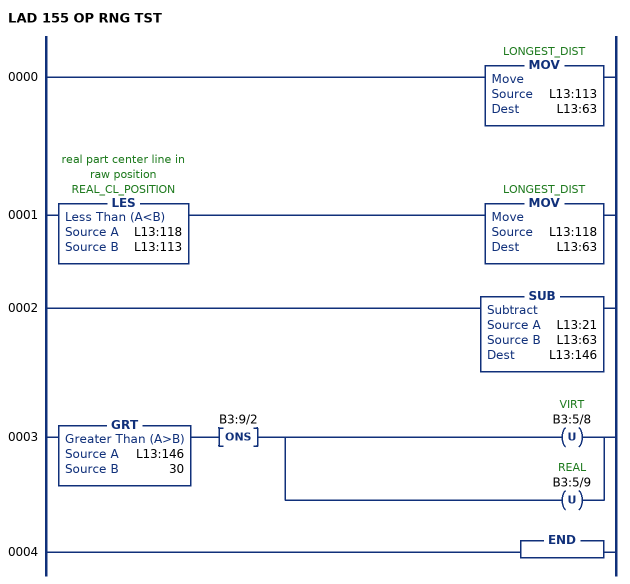
% Rung: 0 %
SOR MOV L13:113 L13:63 EOR
%   L13:113  VERTUAL_CL_POSITION  "virtual part center line transfer from the bottom in raw position" %
%   L13:63  LONGEST_DIST %
% Rung: 1 %
SOR LES L13:118 L13:113 MOV L13:118 L13:63 EOR
%   L13:118  REAL_CL_POSITION  "real part center line in raw position" %
%   L13:113  VERTUAL_CL_POSITION  "virtual part center line transfer from the bottom in raw position" %
%   L13:63  LONGEST_DIST %
% Rung: 2 %
SOR SUB L13:21 L13:63 L13:146 EOR
%   L13:21  TOP_POSITION %
%   L13:63  LONGEST_DIST %
% Rung: 3 %
SOR GRT L13:146 30 ONS B3:9/2 BST OTU B3:5/8 NXB OTU B3:5/9 BND EOR
%   B3:5/8  VIRT %
%   B3:5/9  REAL %
% Rung: 4 %
SOR END EOR

LADDER 190 "INS5"
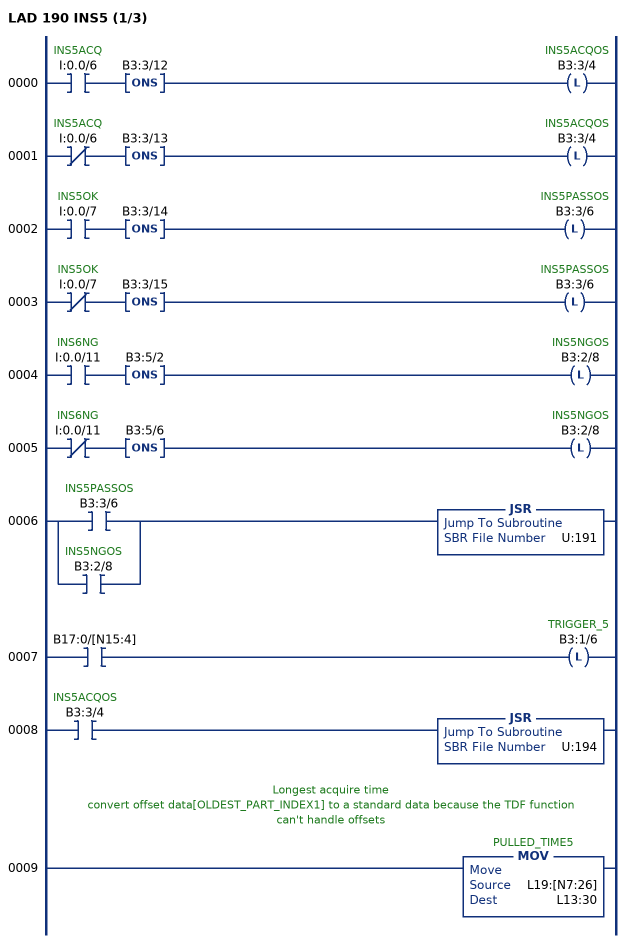
% Rung: 0 %
SOR XIC I:0.0/6 ONS B3:3/12 OTL B3:3/4 EOR
%   I:0.0/6  INS5ACQ %
%   B3:3/4  INS5ACQOS %
% Rung: 1 %
SOR XIO I:0.0/6 ONS B3:3/13 OTL B3:3/4 EOR
%   I:0.0/6  INS5ACQ %
%   B3:3/4  INS5ACQOS %
% Rung: 2 %
SOR XIC I:0.0/7 ONS B3:3/14 OTL B3:3/6 EOR
%   I:0.0/7  INS5OK %
%   B3:3/6  INS5PASSOS %
% Rung: 3 %
SOR XIO I:0.0/7 ONS B3:3/15 OTL B3:3/6 EOR
%   I:0.0/7  INS5OK %
%   B3:3/6  INS5PASSOS %
% Rung: 4 %
SOR XIC I:0.0/11 ONS B3:5/2 OTL B3:2/8 EOR
%   I:0.0/11  INS6NG %
%   B3:2/8  INS5NGOS %
% Rung: 5 %
SOR XIO I:0.0/11 ONS B3:5/6 OTL B3:2/8 EOR
%   I:0.0/11  INS6NG %
%   B3:2/8  INS5NGOS %
% Rung: 6 %
SOR BST XIC B3:3/6 NXB XIC B3:2/8 BND JSR U:191 EOR
%   B3:3/6  INS5PASSOS %
%   B3:2/8  INS5NGOS %
% Rung: 7 %
SOR XIC B17:0/[N15:4] OTL B3:1/6 EOR
%   B17:0  GOOD1 %
%   N15:4  INS_5_TRIG_LOC %
%   B3:1/6  TRIGGER_5 %
% Rung: 8 %
SOR XIC B3:3/4 JSR U:194 EOR
%   B3:3/4  INS5ACQOS %
% Rung: 9 %
% Longest acquire time
% convert offset data[OLDEST_PART_INDEX1] to a standard data because the TDF function can't handle offsets %
SOR MOV L19:[N7:26] L13:30 EOR
%   N7:26  OLDEST_PART_INDEX5 %
%   L13:30  PULLED_TIME5 %

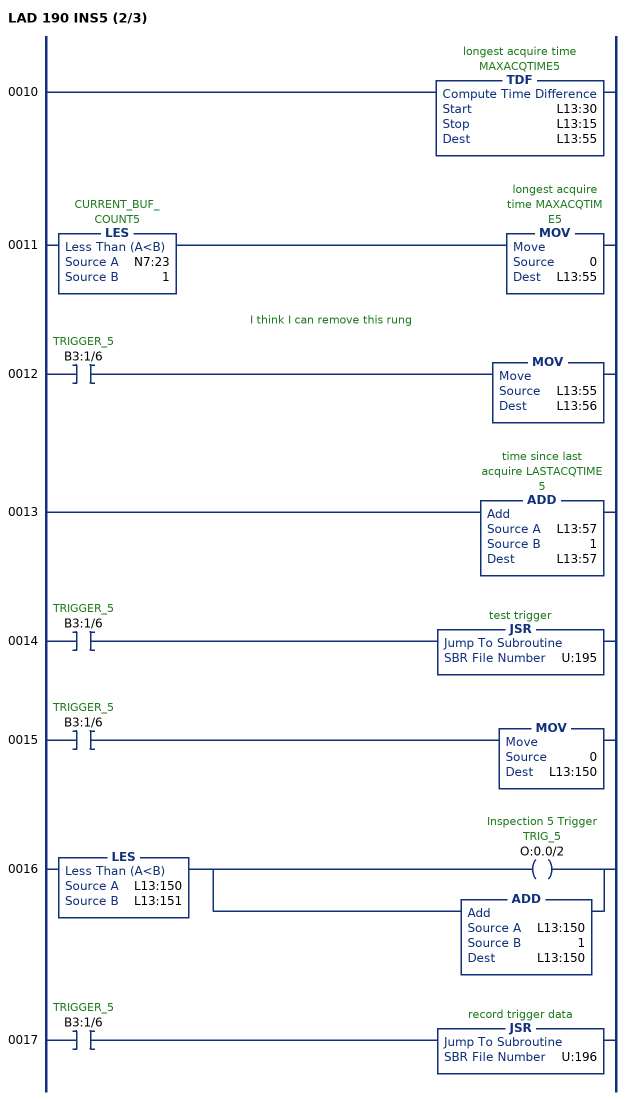
% Rung: 10 %
SOR TDF L13:30 L13:15 L13:55 EOR
%   L13:30  PULLED_TIME5 %
%   L13:15  TOP_TIME %
%   L13:55  MAXACQTIME5  "longest acquire time" %
% Rung: 11 %
SOR LES N7:23 1 MOV 0 L13:55 EOR
%   N7:23  CURRENT_BUF_COUNT5 %
%   L13:55  MAXACQTIME5  "longest acquire time" %
% Rung: 12 %
% I think I can remove this rung %
SOR XIC B3:1/6 MOV L13:55 L13:56 EOR
%   B3:1/6  TRIGGER_5 %
%   L13:55  MAXACQTIME5  "longest acquire time" %
% Rung: 13 %
SOR ADD L13:57 1 L13:57 EOR
%   L13:57  LASTACQTIME5  "time since last acquire" %
% Rung: 14 %
SOR XIC B3:1/6 JSR U:195 EOR
%   B3:1/6  TRIGGER_5 %
%   U:195  "test trigger" %
% Rung: 15 %
SOR XIC B3:1/6 MOV 0 L13:150 EOR
%   B3:1/6  TRIGGER_5 %
% Rung: 16 %
SOR LES L13:150 L13:151 BST OTE O:0.0/2 NXB ADD L13:150 1 L13:150 BND EOR
%   O:0.0/2  TRIG_5  "Inspection 5 Trigger" %
% Rung: 17 %
SOR XIC B3:1/6 JSR U:196 EOR
%   B3:1/6  TRIGGER_5 %
%   U:196  "record trigger data" %

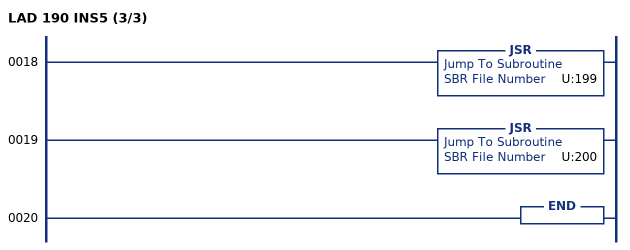
% Rung: 18 %
SOR JSR U:199 EOR
% Rung: 19 %
SOR JSR U:200 EOR
% Rung: 20 %
SOR END EOR

LADDER 191 "INS5RESULT"
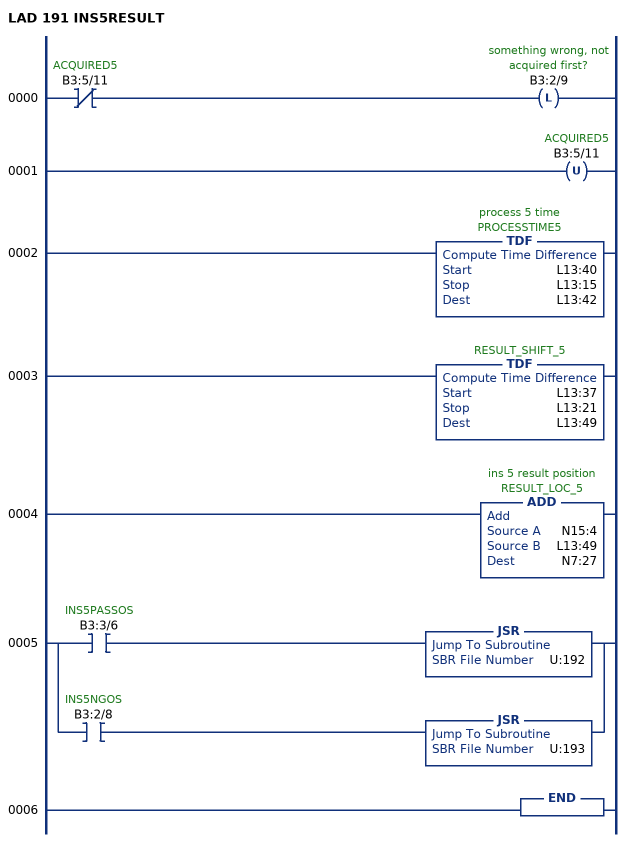
% Rung: 0 %
SOR XIO B3:5/11 OTL B3:2/9 EOR
%   B3:5/11  ACQUIRED5 %
%   B3:2/9  "something wrong, not acquired first?" %
% Rung: 1 %
SOR OTU B3:5/11 EOR
%   B3:5/11  ACQUIRED5 %
% Rung: 2 %
SOR TDF L13:40 L13:15 L13:42 EOR
%   L13:40  TIMEOFACQ5  "the time of the last acquire" %
%   L13:15  TOP_TIME %
%   L13:42  PROCESSTIME5  "process 5 time" %
% Rung: 3 %
SOR TDF L13:37 L13:21 L13:49 EOR
%   L13:37  PROCESS_START_POS_5 %
%   L13:21  TOP_POSITION %
%   L13:49  RESULT_SHIFT_5 %
% Rung: 4 %
SOR ADD N15:4 L13:49 N7:27 EOR
%   N15:4  INS_5_TRIG_LOC %
%   L13:49  RESULT_SHIFT_5 %
%   N7:27  RESULT_LOC_5  "ins 5 result position" %
% Rung: 5 %
SOR BST XIC B3:3/6 JSR U:192 NXB XIC B3:2/8 JSR U:193 BND EOR
%   B3:3/6  INS5PASSOS %
%   B3:2/8  INS5NGOS %
% Rung: 6 %
SOR END EOR

LADDER 192 "INS5PASS"
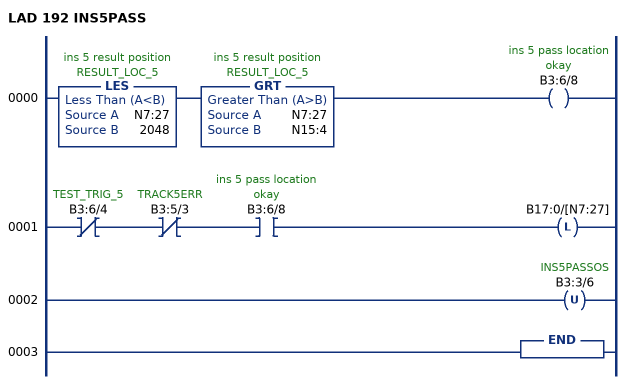
% Rung: 0 %
SOR LES N7:27 2048 GRT N7:27 N15:4 OTE B3:6/8 EOR
%   N7:27  RESULT_LOC_5  "ins 5 result position" %
%   N15:4  INS_5_TRIG_LOC %
%   B3:6/8  "ins 5 pass location okay" %
% Rung: 1 %
SOR XIO B3:6/4 XIO B3:5/3 XIC B3:6/8 OTL B17:0/[N7:27] EOR
%   B3:6/4  TEST_TRIG_5 %
%   B3:5/3  TRACK5ERR %
%   B3:6/8  "ins 5 pass location okay" %
%   B17:0  GOOD1 %
%   N7:27  RESULT_LOC_5  "ins 5 result position" %
% Rung: 2 %
SOR OTU B3:3/6 EOR
%   B3:3/6  INS5PASSOS %
% Rung: 3 %
SOR END EOR

LADDER 193 "INS5FAIL"
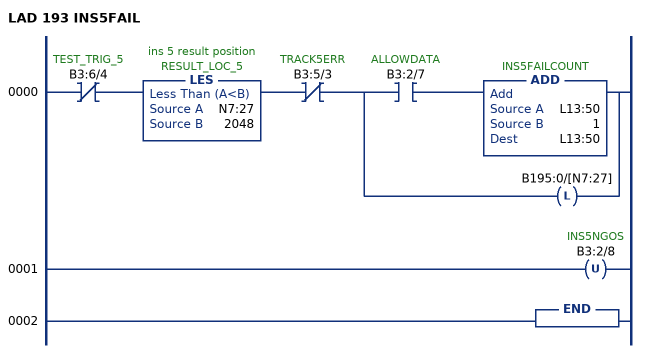
% Rung: 0 %
SOR XIO B3:6/4 LES N7:27 2048 XIO B3:5/3 BST XIC B3:2/7 ADD L13:50 1 L13:50 NXB OTL B195:0/[N7:27] BND EOR
%   B3:6/4  TEST_TRIG_5 %
%   N7:27  RESULT_LOC_5  "ins 5 result position" %
%   B3:5/3  TRACK5ERR %
%   B3:2/7  ALLOWDATA %
%   L13:50  INS5FAILCOUNT %
%   B195:0  TOP_NG %
% Rung: 1 %
SOR OTU B3:2/8 EOR
%   B3:2/8  INS5NGOS %
% Rung: 2 %
SOR END EOR

LADDER 194 "INS5ACQ"
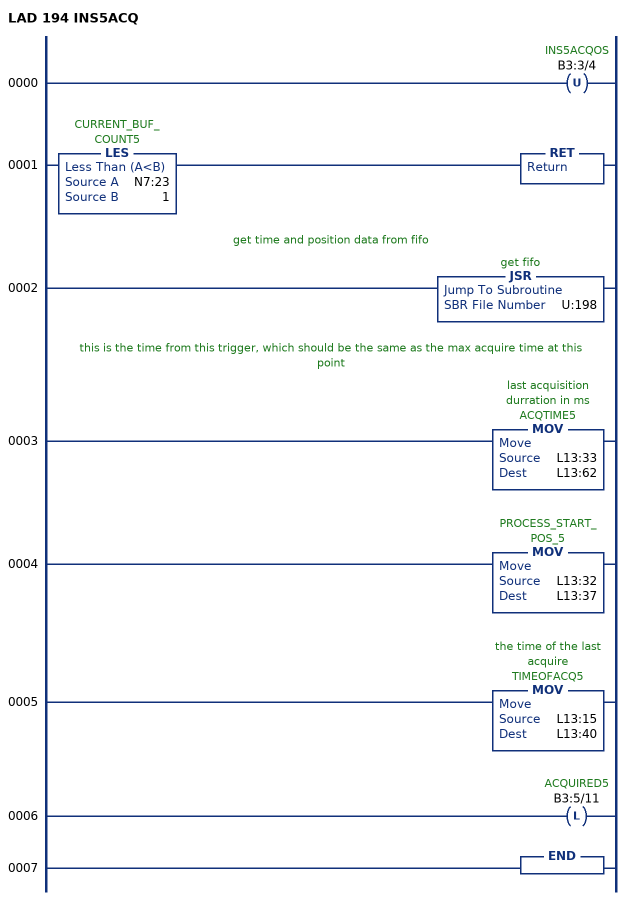
% Rung: 0 %
SOR OTU B3:3/4 EOR
%   B3:3/4  INS5ACQOS %
% Rung: 1 %
SOR LES N7:23 1 RET EOR
%   N7:23  CURRENT_BUF_COUNT5 %
% Rung: 2 %
% get time and position data from fifo %
SOR JSR U:198 EOR
%   U:198  "get fifo" %
% Rung: 3 %
% this is the time from this trigger, which should be the same as the max acquire time at this point %
SOR MOV L13:33 L13:62 EOR
%   L13:33  TIME_SPAN5 %
%   L13:62  ACQTIME5  "last acquisition durration in ms" %
% Rung: 4 %
SOR MOV L13:32 L13:37 EOR
%   L13:32  PULLED_POSITION5 %
%   L13:37  PROCESS_START_POS_5 %
% Rung: 5 %
SOR MOV L13:15 L13:40 EOR
%   L13:15  TOP_TIME %
%   L13:40  TIMEOFACQ5  "the time of the last acquire" %
% Rung: 6 %
SOR OTL B3:5/11 EOR
%   B3:5/11  ACQUIRED5 %
% Rung: 7 %
SOR END EOR

LADDER 195 "Q5TIMETEST"
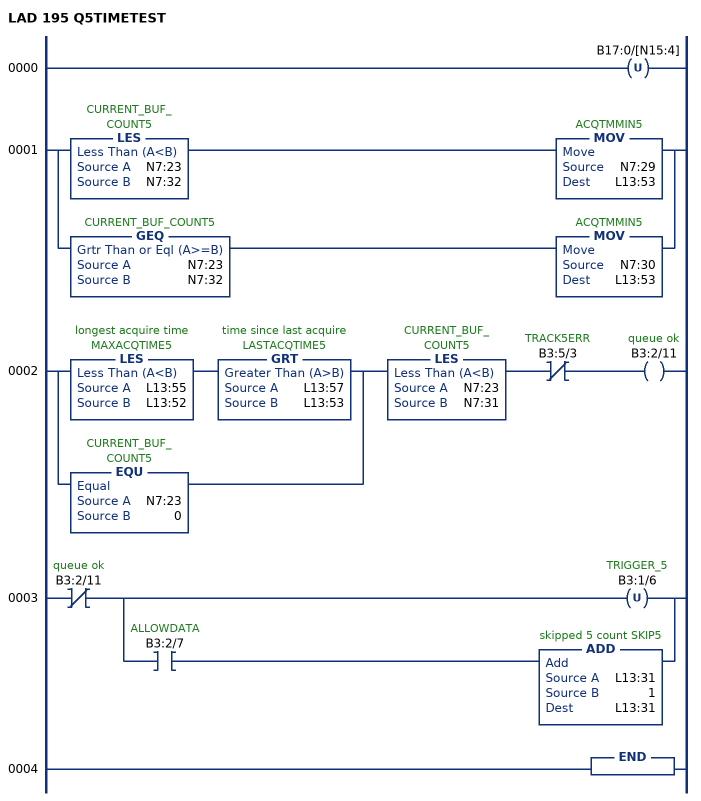
% Rung: 0 %
SOR OTU B17:0/[N15:4] EOR
%   B17:0  GOOD1 %
%   N15:4  INS_5_TRIG_LOC %
% Rung: 1 %
SOR BST LES N7:23 N7:32 MOV N7:29 L13:53 NXB GEQ N7:23 N7:32 MOV N7:30 L13:53 BND EOR
%   N7:23  CURRENT_BUF_COUNT5 %
%   N7:32  BUF_CAM_LIMIT %
%   N7:29  CAM_BUF_ACQ_TM %
%   L13:53  ACQTMMIN5 %
%   N7:30  PC_BUF_ACQ_TM %
% Rung: 2 %
SOR BST LES L13:55 L13:52 GRT L13:57 L13:53 NXB EQU N7:23 0 BND LES N7:23 N7:31 XIO B3:5/3 OTE B3:2/11 EOR
%   L13:55  MAXACQTIME5  "longest acquire time" %
%   L13:52  ACQTIMELIMIT %
%   L13:57  LASTACQTIME5  "time since last acquire" %
%   L13:53  ACQTMMIN5 %
%   N7:23  CURRENT_BUF_COUNT5 %
%   N7:31  MAX_BUFF_CT  "maximum buffers" %
%   B3:5/3  TRACK5ERR %
%   B3:2/11  "queue ok" %
% Rung: 3 %
SOR XIO B3:2/11 BST OTU B3:1/6 NXB XIC B3:2/7 ADD L13:31 1 L13:31 BND EOR
%   B3:2/11  "queue ok" %
%   B3:1/6  TRIGGER_5 %
%   B3:2/7  ALLOWDATA %
%   L13:31  SKIP5  "skipped 5 count" %
% Rung: 4 %
SOR END EOR

LADDER 196 "INS5TRIG"
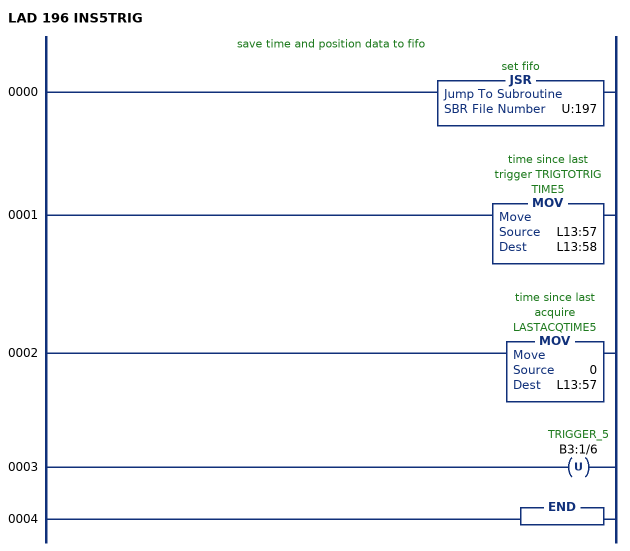
% Rung: 0 %
% save time and position data to fifo %
SOR JSR U:197 EOR
%   U:197  "set fifo" %
% Rung: 1 %
SOR MOV L13:57 L13:58 EOR
%   L13:57  LASTACQTIME5  "time since last acquire" %
%   L13:58  TRIGTOTRIGTIME5  "time since last trigger" %
% Rung: 2 %
SOR MOV 0 L13:57 EOR
%   L13:57  LASTACQTIME5  "time since last acquire" %
% Rung: 3 %
SOR OTU B3:1/6 EOR
%   B3:1/6  TRIGGER_5 %
% Rung: 4 %
SOR END EOR

LADDER 197 "FIFO5SET"
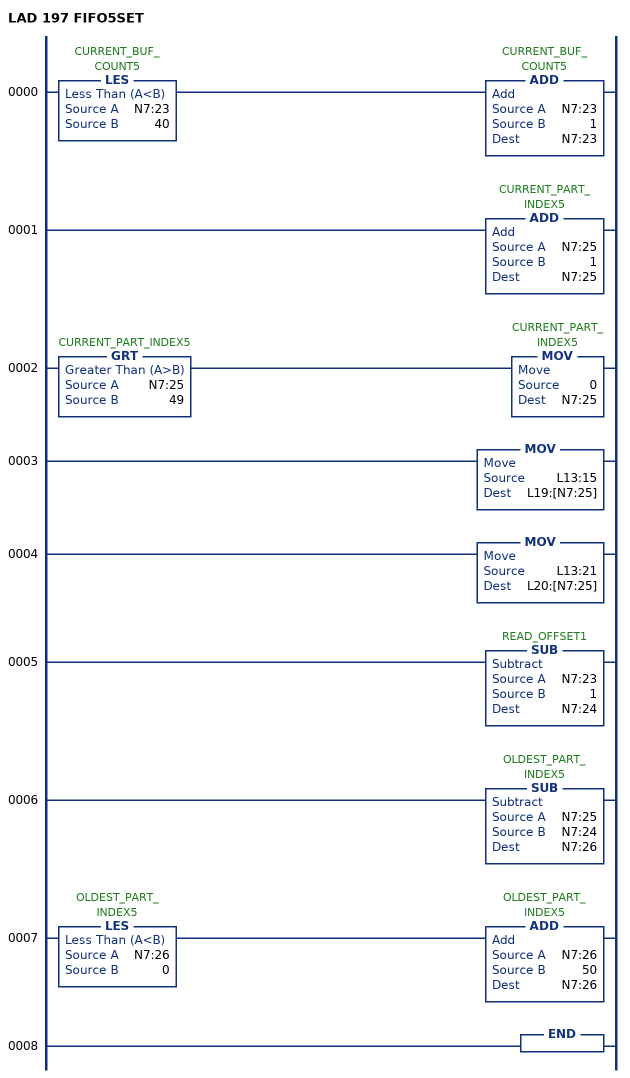
% Rung: 0 %
SOR LES N7:23 40 ADD N7:23 1 N7:23 EOR
%   N7:23  CURRENT_BUF_COUNT5 %
% Rung: 1 %
SOR ADD N7:25 1 N7:25 EOR
%   N7:25  CURRENT_PART_INDEX5 %
% Rung: 2 %
SOR GRT N7:25 49 MOV 0 N7:25 EOR
%   N7:25  CURRENT_PART_INDEX5 %
% Rung: 3 %
SOR MOV L13:15 L19:[N7:25] EOR
%   L13:15  TOP_TIME %
%   N7:25  CURRENT_PART_INDEX5 %
% Rung: 4 %
SOR MOV L13:21 L20:[N7:25] EOR
%   L13:21  TOP_POSITION %
%   N7:25  CURRENT_PART_INDEX5 %
% Rung: 5 %
SOR SUB N7:23 1 N7:24 EOR
%   N7:23  CURRENT_BUF_COUNT5 %
%   N7:24  "READ_OFFSET1" %
% Rung: 6 %
SOR SUB N7:25 N7:24 N7:26 EOR
%   N7:25  CURRENT_PART_INDEX5 %
%   N7:24  "READ_OFFSET1" %
%   N7:26  OLDEST_PART_INDEX5 %
% Rung: 7 %
SOR LES N7:26 0 ADD N7:26 50 N7:26 EOR
%   N7:26  OLDEST_PART_INDEX5 %
% Rung: 8 %
SOR END EOR

LADDER 198 "FIFO5GET"
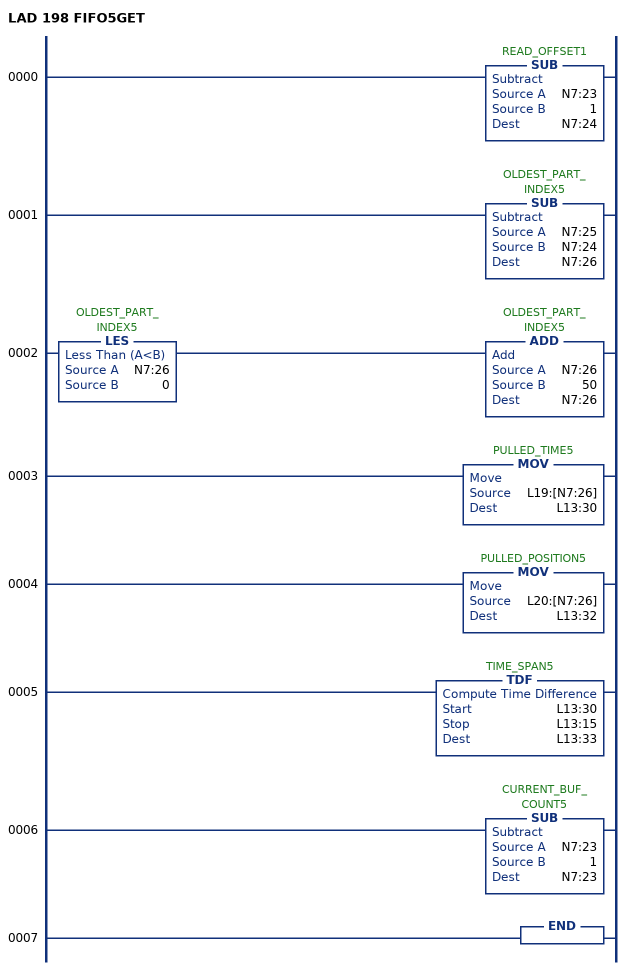
% Rung: 0 %
SOR SUB N7:23 1 N7:24 EOR
%   N7:23  CURRENT_BUF_COUNT5 %
%   N7:24  "READ_OFFSET1" %
% Rung: 1 %
SOR SUB N7:25 N7:24 N7:26 EOR
%   N7:25  CURRENT_PART_INDEX5 %
%   N7:24  "READ_OFFSET1" %
%   N7:26  OLDEST_PART_INDEX5 %
% Rung: 2 %
SOR LES N7:26 0 ADD N7:26 50 N7:26 EOR
%   N7:26  OLDEST_PART_INDEX5 %
% Rung: 3 %
SOR MOV L19:[N7:26] L13:30 EOR
%   N7:26  OLDEST_PART_INDEX5 %
%   L13:30  PULLED_TIME5 %
% Rung: 4 %
SOR MOV L20:[N7:26] L13:32 EOR
%   N7:26  OLDEST_PART_INDEX5 %
%   L13:32  PULLED_POSITION5 %
% Rung: 5 %
SOR TDF L13:30 L13:15 L13:33 EOR
%   L13:30  PULLED_TIME5 %
%   L13:15  TOP_TIME %
%   L13:33  TIME_SPAN5 %
% Rung: 6 %
SOR SUB N7:23 1 N7:23 EOR
%   N7:23  CURRENT_BUF_COUNT5 %
% Rung: 7 %
SOR END EOR

LADDER 199 "INSDATA5"
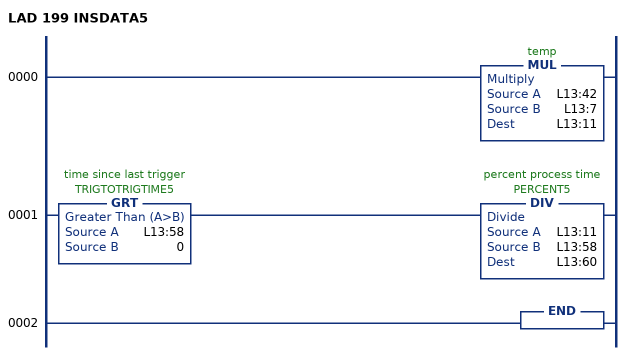
% Rung: 0 %
SOR MUL L13:42 L13:7 L13:11 EOR
%   L13:42  PROCESSTIME5  "process 5 time" %
%   L13:7  PERCENT_MULTIPLYER %
%   L13:11  "temp" %
% Rung: 1 %
SOR GRT L13:58 0 DIV L13:11 L13:58 L13:60 EOR
%   L13:58  TRIGTOTRIGTIME5  "time since last trigger" %
%   L13:11  "temp" %
%   L13:60  PERCENT5  "percent process time" %
% Rung: 2 %
SOR END EOR

LADDER 200 "TESTFAULT5"
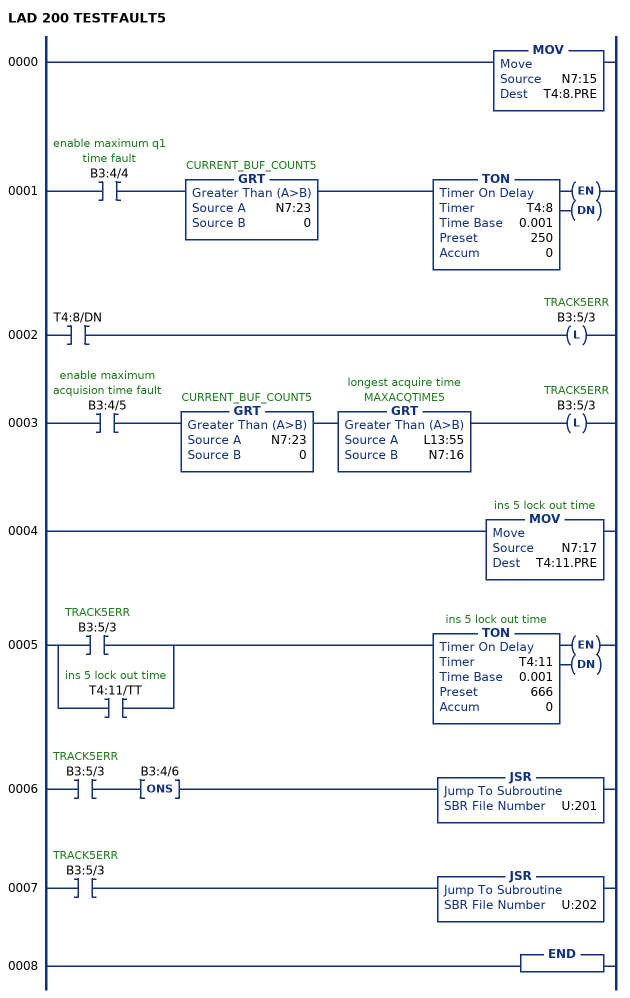
% Rung: 0 %
SOR MOV N7:15 T4:8.PRE EOR
%   N7:15  "max allowed ms time for q to be above 1 if safe fault is used" %
% Rung: 1 %
SOR XIC B3:4/4 GRT N7:23 0 TON T4:8 0.001 250 0 EOR
%   B3:4/4  "enable maximum q1 time fault" %
%   N7:23  CURRENT_BUF_COUNT5 %
% Rung: 2 %
SOR XIC T4:8/DN OTL B3:5/3 EOR
%   B3:5/3  TRACK5ERR %
% Rung: 3 %
SOR XIC B3:4/5 GRT N7:23 0 GRT L13:55 N7:16 OTL B3:5/3 EOR
%   B3:4/5  "enable maximum acquision time fault" %
%   N7:23  CURRENT_BUF_COUNT5 %
%   L13:55  MAXACQTIME5  "longest acquire time" %
%   N7:16  ACQUIRE_TIME_LIMIT  "maximum of the longest acquire time allowed if maximum acquire time fault is enabled" %
%   B3:5/3  TRACK5ERR %
% Rung: 4 %
SOR MOV N7:17 T4:11.PRE EOR
%   N7:17  "ms time setting to lock out inspection to give all pending images a chance to clear" %
%   T4:11  "ins 5 lock out time" %
% Rung: 5 %
SOR BST XIC B3:5/3 NXB XIC T4:11/TT BND TON T4:11 0.001 666 0 EOR
%   B3:5/3  TRACK5ERR %
%   T4:11  "ins 5 lock out time" %
% Rung: 6 %
SOR XIC B3:5/3 ONS B3:4/6 JSR U:201 EOR
%   B3:5/3  TRACK5ERR %
% Rung: 7 %
SOR XIC B3:5/3 JSR U:202 EOR
%   B3:5/3  TRACK5ERR %
% Rung: 8 %
SOR END EOR

LADDER 201 "INS5FIX1"
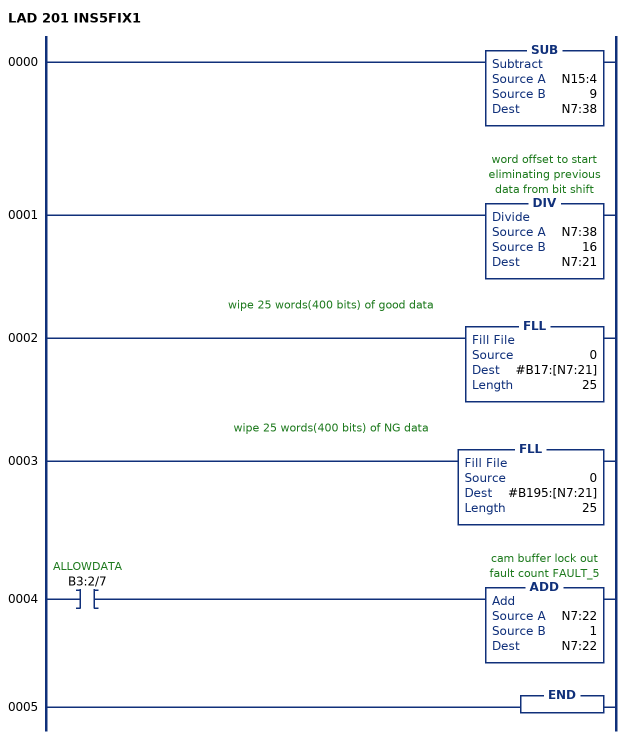
% Rung: 0 %
SOR SUB N15:4 9 N7:38 EOR
%   N15:4  INS_5_TRIG_LOC %
% Rung: 1 %
SOR DIV N7:38 16 N7:21 EOR
%   N7:21  "word offset to start eliminating previous data from bit shift" %
% Rung: 2 %
% wipe 25 words(400 bits) of good data %
SOR FLL 0 #B17:[N7:21] 25 EOR
%   N7:21  "word offset to start eliminating previous data from bit shift" %
% Rung: 3 %
% wipe 25 words(400 bits) of NG data %
SOR FLL 0 #B195:[N7:21] 25 EOR
%   N7:21  "word offset to start eliminating previous data from bit shift" %
% Rung: 4 %
SOR XIC B3:2/7 ADD N7:22 1 N7:22 EOR
%   B3:2/7  ALLOWDATA %
%   N7:22  FAULT_5  "cam buffer lock out fault count" %
% Rung: 5 %
SOR END EOR

LADDER 202 "INS5FIX2"
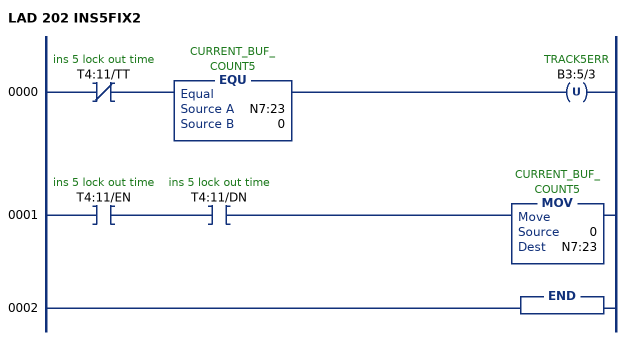
% Rung: 0 %
SOR XIO T4:11/TT EQU N7:23 0 OTU B3:5/3 EOR
%   T4:11  "ins 5 lock out time" %
%   N7:23  CURRENT_BUF_COUNT5 %
%   B3:5/3  TRACK5ERR %
% Rung: 1 %
SOR XIC T4:11/EN XIC T4:11/DN MOV 0 N7:23 EOR
%   T4:11  "ins 5 lock out time" %
%   N7:23  CURRENT_BUF_COUNT5 %
% Rung: 2 %
SOR END EOR

LADDER 204 "INS6"
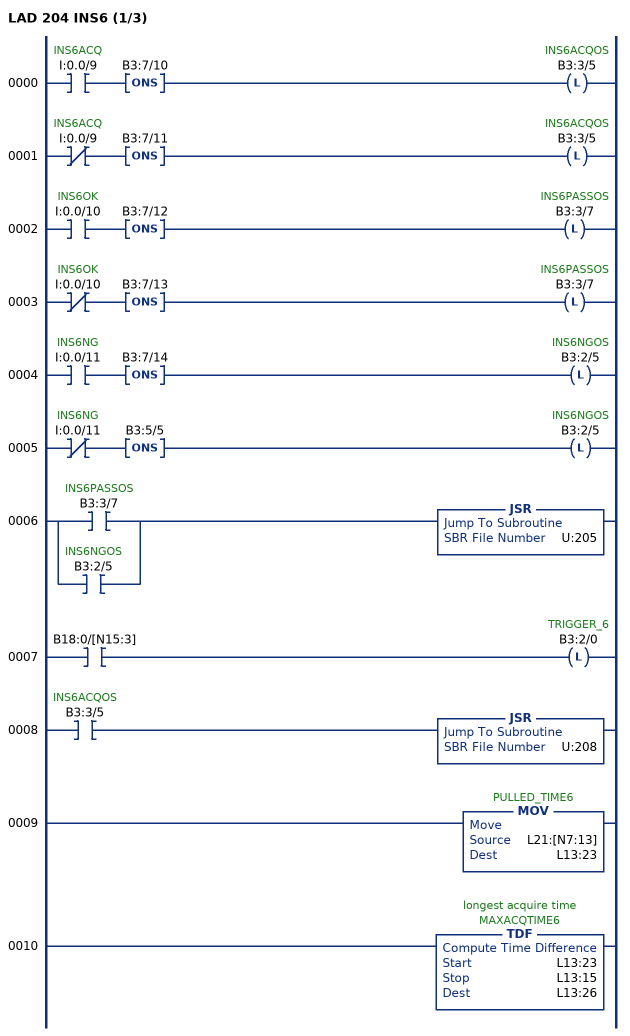
% Rung: 0 %
SOR XIC I:0.0/9 ONS B3:7/10 OTL B3:3/5 EOR
%   I:0.0/9  INS6ACQ %
%   B3:3/5  INS6ACQOS %
% Rung: 1 %
SOR XIO I:0.0/9 ONS B3:7/11 OTL B3:3/5 EOR
%   I:0.0/9  INS6ACQ %
%   B3:3/5  INS6ACQOS %
% Rung: 2 %
SOR XIC I:0.0/10 ONS B3:7/12 OTL B3:3/7 EOR
%   I:0.0/10  INS6OK %
%   B3:3/7  INS6PASSOS %
% Rung: 3 %
SOR XIO I:0.0/10 ONS B3:7/13 OTL B3:3/7 EOR
%   I:0.0/10  INS6OK %
%   B3:3/7  INS6PASSOS %
% Rung: 4 %
SOR XIC I:0.0/11 ONS B3:7/14 OTL B3:2/5 EOR
%   I:0.0/11  INS6NG %
%   B3:2/5  INS6NGOS %
% Rung: 5 %
SOR XIO I:0.0/11 ONS B3:5/5 OTL B3:2/5 EOR
%   I:0.0/11  INS6NG %
%   B3:2/5  INS6NGOS %
% Rung: 6 %
SOR BST XIC B3:3/7 NXB XIC B3:2/5 BND JSR U:205 EOR
%   B3:3/7  INS6PASSOS %
%   B3:2/5  INS6NGOS %
% Rung: 7 %
SOR XIC B18:0/[N15:3] OTL B3:2/0 EOR
%   B18:0  GOOD2 %
%   N15:3  INS_6_TRIG_LOC %
%   B3:2/0  TRIGGER_6 %
% Rung: 8 %
SOR XIC B3:3/5 JSR U:208 EOR
%   B3:3/5  INS6ACQOS %
% Rung: 9 %
SOR MOV L21:[N7:13] L13:23 EOR
%   N7:13  OLDEST_PART_INDEX6 %
%   L13:23  PULLED_TIME6 %
% Rung: 10 %
SOR TDF L13:23 L13:15 L13:26 EOR
%   L13:23  PULLED_TIME6 %
%   L13:15  TOP_TIME %
%   L13:26  MAXACQTIME6  "longest acquire time" %

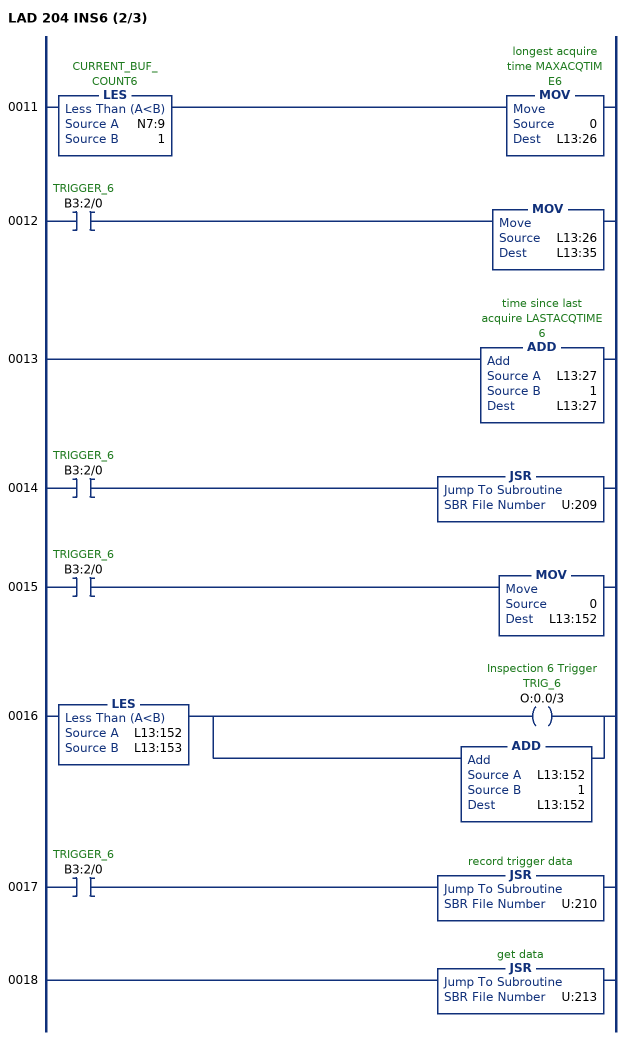
% Rung: 11 %
SOR LES N7:9 1 MOV 0 L13:26 EOR
%   N7:9  CURRENT_BUF_COUNT6 %
%   L13:26  MAXACQTIME6  "longest acquire time" %
% Rung: 12 %
SOR XIC B3:2/0 MOV L13:26 L13:35 EOR
%   B3:2/0  TRIGGER_6 %
%   L13:26  MAXACQTIME6  "longest acquire time" %
% Rung: 13 %
SOR ADD L13:27 1 L13:27 EOR
%   L13:27  LASTACQTIME6  "time since last acquire" %
% Rung: 14 %
SOR XIC B3:2/0 JSR U:209 EOR
%   B3:2/0  TRIGGER_6 %
% Rung: 15 %
SOR XIC B3:2/0 MOV 0 L13:152 EOR
%   B3:2/0  TRIGGER_6 %
% Rung: 16 %
SOR LES L13:152 L13:153 BST OTE O:0.0/3 NXB ADD L13:152 1 L13:152 BND EOR
%   O:0.0/3  TRIG_6  "Inspection 6 Trigger" %
% Rung: 17 %
SOR XIC B3:2/0 JSR U:210 EOR
%   B3:2/0  TRIGGER_6 %
%   U:210  "record trigger data" %
% Rung: 18 %
SOR JSR U:213 EOR
%   U:213  "get data" %

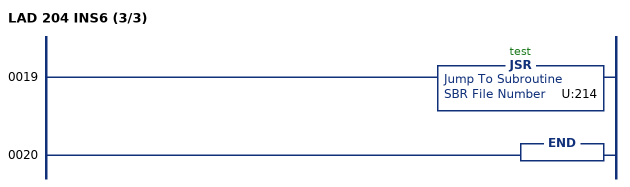
% Rung: 19 %
SOR JSR U:214 EOR
%   U:214  "test" %
% Rung: 20 %
SOR END EOR

LADDER 205 "INS6RESULT"
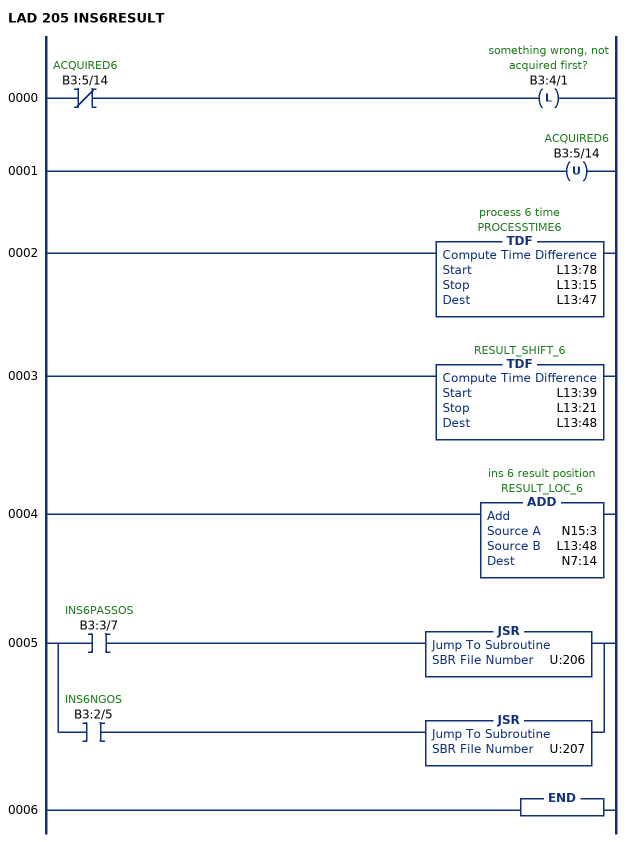
% Rung: 0 %
SOR XIO B3:5/14 OTL B3:4/1 EOR
%   B3:5/14  ACQUIRED6 %
%   B3:4/1  "something wrong, not acquired first?" %
% Rung: 1 %
SOR OTU B3:5/14 EOR
%   B3:5/14  ACQUIRED6 %
% Rung: 2 %
SOR TDF L13:78 L13:15 L13:47 EOR
%   L13:78  TIMEOFACQ6  "the time of the last acquire" %
%   L13:15  TOP_TIME %
%   L13:47  PROCESSTIME6  "process 6 time" %
% Rung: 3 %
SOR TDF L13:39 L13:21 L13:48 EOR
%   L13:39  PROCESS_START_POS_6 %
%   L13:21  TOP_POSITION %
%   L13:48  RESULT_SHIFT_6 %
% Rung: 4 %
SOR ADD N15:3 L13:48 N7:14 EOR
%   N15:3  INS_6_TRIG_LOC %
%   L13:48  RESULT_SHIFT_6 %
%   N7:14  RESULT_LOC_6  "ins 6 result position" %
% Rung: 5 %
SOR BST XIC B3:3/7 JSR U:206 NXB XIC B3:2/5 JSR U:207 BND EOR
%   B3:3/7  INS6PASSOS %
%   B3:2/5  INS6NGOS %
% Rung: 6 %
SOR END EOR

LADDER 206 "INS6PASS"
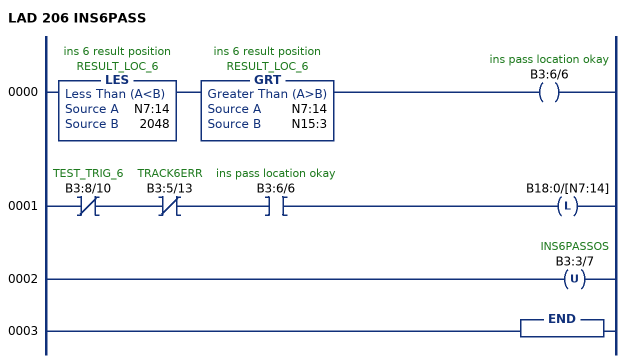
% Rung: 0 %
SOR LES N7:14 2048 GRT N7:14 N15:3 OTE B3:6/6 EOR
%   N7:14  RESULT_LOC_6  "ins 6 result position" %
%   N15:3  INS_6_TRIG_LOC %
%   B3:6/6  "ins pass location okay" %
% Rung: 1 %
SOR XIO B3:8/10 XIO B3:5/13 XIC B3:6/6 OTL B18:0/[N7:14] EOR
%   B3:8/10  TEST_TRIG_6 %
%   B3:5/13  TRACK6ERR %
%   B3:6/6  "ins pass location okay" %
%   B18:0  GOOD2 %
%   N7:14  RESULT_LOC_6  "ins 6 result position" %
% Rung: 2 %
SOR OTU B3:3/7 EOR
%   B3:3/7  INS6PASSOS %
% Rung: 3 %
SOR END EOR

LADDER 207 "INS6FAIL"
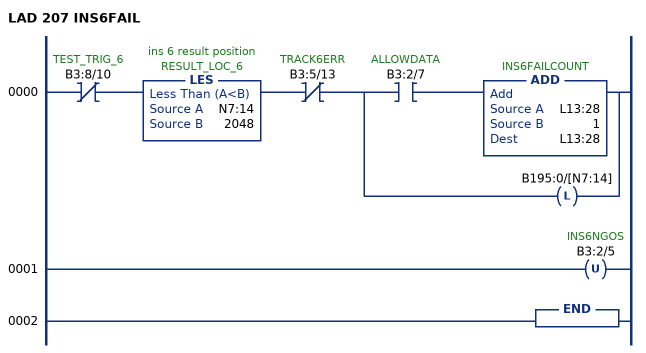
% Rung: 0 %
SOR XIO B3:8/10 LES N7:14 2048 XIO B3:5/13 BST XIC B3:2/7 ADD L13:28 1 L13:28 NXB OTL B195:0/[N7:14] BND EOR
%   B3:8/10  TEST_TRIG_6 %
%   N7:14  RESULT_LOC_6  "ins 6 result position" %
%   B3:5/13  TRACK6ERR %
%   B3:2/7  ALLOWDATA %
%   L13:28  INS6FAILCOUNT %
%   B195:0  TOP_NG %
% Rung: 1 %
SOR OTU B3:2/5 EOR
%   B3:2/5  INS6NGOS %
% Rung: 2 %
SOR END EOR

LADDER 208 "INS6ACQ"
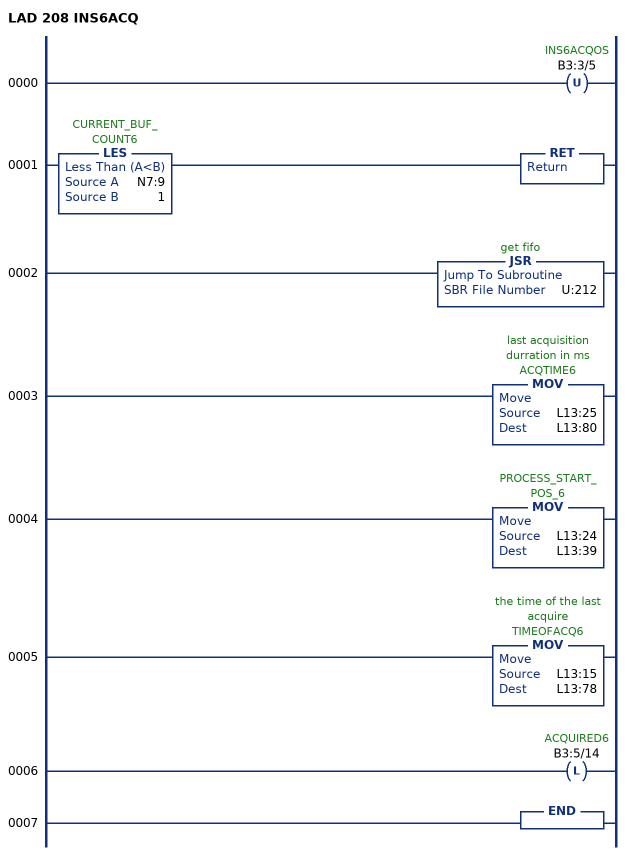
% Rung: 0 %
SOR OTU B3:3/5 EOR
%   B3:3/5  INS6ACQOS %
% Rung: 1 %
SOR LES N7:9 1 RET EOR
%   N7:9  CURRENT_BUF_COUNT6 %
% Rung: 2 %
SOR JSR U:212 EOR
%   U:212  "get fifo" %
% Rung: 3 %
SOR MOV L13:25 L13:80 EOR
%   L13:25  TIME_SPAN6 %
%   L13:80  ACQTIME6  "last acquisition durration in ms" %
% Rung: 4 %
SOR MOV L13:24 L13:39 EOR
%   L13:24  PULLED_POSITION6 %
%   L13:39  PROCESS_START_POS_6 %
% Rung: 5 %
SOR MOV L13:15 L13:78 EOR
%   L13:15  TOP_TIME %
%   L13:78  TIMEOFACQ6  "the time of the last acquire" %
% Rung: 6 %
SOR OTL B3:5/14 EOR
%   B3:5/14  ACQUIRED6 %
% Rung: 7 %
SOR END EOR

LADDER 209 "Q6TIMETEST"
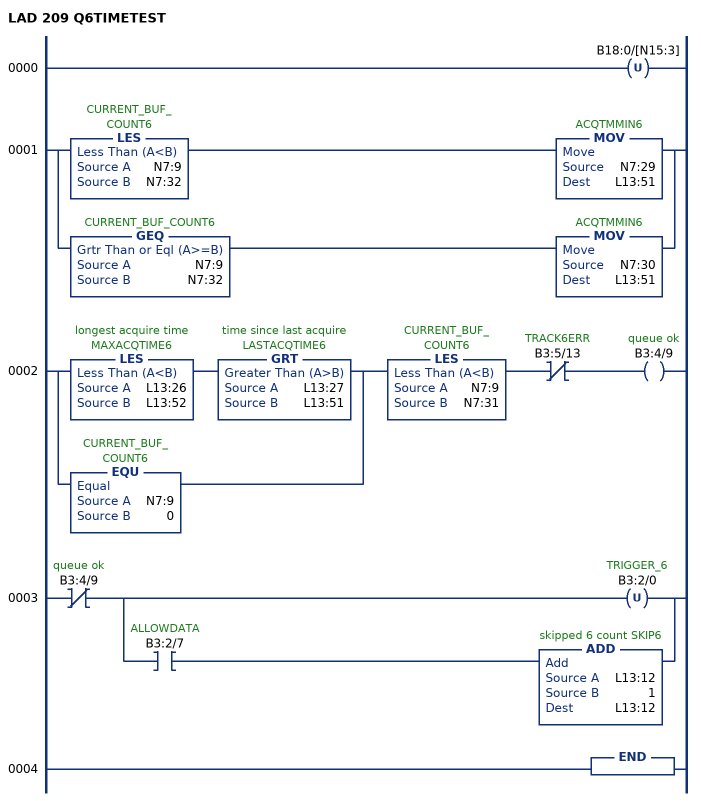
% Rung: 0 %
SOR OTU B18:0/[N15:3] EOR
%   B18:0  GOOD2 %
%   N15:3  INS_6_TRIG_LOC %
% Rung: 1 %
SOR BST LES N7:9 N7:32 MOV N7:29 L13:51 NXB GEQ N7:9 N7:32 MOV N7:30 L13:51 BND EOR
%   N7:9  CURRENT_BUF_COUNT6 %
%   N7:32  BUF_CAM_LIMIT %
%   N7:29  CAM_BUF_ACQ_TM %
%   L13:51  ACQTMMIN6 %
%   N7:30  PC_BUF_ACQ_TM %
% Rung: 2 %
SOR BST LES L13:26 L13:52 GRT L13:27 L13:51 NXB EQU N7:9 0 BND LES N7:9 N7:31 XIO B3:5/13 OTE B3:4/9 EOR
%   L13:26  MAXACQTIME6  "longest acquire time" %
%   L13:52  ACQTIMELIMIT %
%   L13:27  LASTACQTIME6  "time since last acquire" %
%   L13:51  ACQTMMIN6 %
%   N7:9  CURRENT_BUF_COUNT6 %
%   N7:31  MAX_BUFF_CT  "maximum buffers" %
%   B3:5/13  TRACK6ERR %
%   B3:4/9  "queue ok" %
% Rung: 3 %
SOR XIO B3:4/9 BST OTU B3:2/0 NXB XIC B3:2/7 ADD L13:12 1 L13:12 BND EOR
%   B3:4/9  "queue ok" %
%   B3:2/0  TRIGGER_6 %
%   B3:2/7  ALLOWDATA %
%   L13:12  SKIP6  "skipped 6 count" %
% Rung: 4 %
SOR END EOR

LADDER 210 "INS6TRIG"
